(* IEC 61131-3 sources: progetto2711AX/src, 3 files *)

(* ---- somma.st ---- *)
NAMESPACE myLibrary

FUNCTION mySomma : INT
    VAR_INPUT
        a : INT;
        b : INT;
    END_VAR

    VAR
        {S7.extern=ReadOnly}
        myStat : REAL;
    END_VAR

    mySomma := a + b;

    myStat := mySomma + 7;

END_FUNCTION

END_NAMESPACE

(* ---- library.st ---- *)
NAMESPACE ExampleClassLib
    CLASS Belt
       METHOD PUBLIC RunForward ; END_METHOD
       METHOD PUBLIC RunBackward ; END_METHOD
       METHOD PUBLIC Stop ; END_METHOD
    END_CLASS

    CLASS ABSTRACT Conveyor
       METHOD PUBLIC ABSTRACT Run END_METHOD
       METHOD PUBLIC ABSTRACT Stop END_METHOD
    END_CLASS

    CLASS OneBeltConveyor EXTENDS Conveyor
       VAR PUBLIC
          belt : REF_TO Belt;
       END_VAR

       METHOD PUBLIC OVERRIDE Run
         belt^.RunForward();
       END_METHOD

       METHOD PUBLIC OVERRIDE Stop
          belt^.Stop();
       END_METHOD
    END_CLASS

    CLASS TwoBeltConveyor EXTENDS Conveyor
       VAR PUBLIC
          belt1 : REF_TO Belt;
          belt2 : REF_TO Belt;
       END_VAR

       METHOD PUBLIC OVERRIDE Run
          belt1^.RunForward();
          belt2^.RunBackward();
       END_METHOD

       METHOD PUBLIC OVERRIDE Stop
          belt1^.Stop();
          belt2^.Stop();
       END_METHOD
    END_CLASS
 END_NAMESPACE

 NAMESPACE MotorLibrary

   CLASS PUBLIC Motor
       VAR PRIVATE
           _started : BOOL;
       END_VAR

       VAR PRIVATE

       END_VAR

       METHOD PUBLIC Start : BOOL
           _started := FALSE;
           Start := TRUE;
       END_METHOD
   END_CLASS

END_NAMESPACE

(* ---- wrapper.st ---- *)
NAMESPACE ExampleClassLib.Entry
    ///Questo è il commento della FB
    FUNCTION_BLOCK EquipmentModule1 //Wrapper FB; questo commento non è visibile
       VAR_INPUT
          ///questa è la variabile di Start
          start : BOOL;
          ///questa è la variabile di Stop
          stop : BOOL;
       END_VAR
       VAR // OK, classes can be instantiated in VAR
        {S7.extern=ReadOnly}
          belt1, belt2, belt3 : Belt;
          feed                : OneBeltConveyor;
          transport           : TwoBeltConveyor;
          init                : BOOL := TRUE;
       END_VAR

       IF init THEN
          init := FALSE;
          feed.belt := REF(belt1);
          transport.belt1 := REF(belt2);
          transport.belt2 := REF(belt3);
       END_IF;

       IF start AND NOT stop THEN
          feed.Run();
          // wait 10s
          transport.Run();
       ELSIF stop THEN
          transport.Stop();
          // wait 10s
          feed.Stop();
       END_IF;
    END_FUNCTION_BLOCK
 END_NAMESPACE

 NAMESPACE MotorLibrary

   FUNCTION_BLOCK MotorWrapper
       VAR_INPUT
           start : BOOL;
       END_VAR
       VAR
           m : Motor;
       END_VAR

       IF start THEN
           m.Start();
       END_IF;
   END_FUNCTION_BLOCK

END_NAMESPACE
